FUNCTION_BLOCK ChanRcvBool (* Composite Function Block Type *)
  (* Standard: 61499-2 *)
  (* Version 0.0, 12/6/2023, vaatmar1, nxtControl GmBH, template *)
  PACKAGE Main;
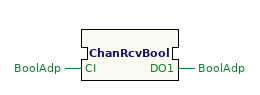
  SOCKETS
    CI : BoolAdp;
  END_SOCKETS
  PLUGS
    DO1 : BoolAdp;
  END_PLUGS
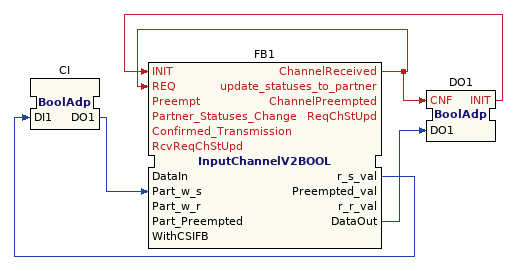
  FBS
    FB1 : InputChannelV2BOOL;
  END_FBS
  EVENT_CONNECTIONS
    DO1.INIT TO FB1.INIT;
    FB1.ChannelReceived TO DO1.CNF;
    FB1.ChannelReceived TO FB1.REQ;
  END_CONNECTIONS
  DATA_CONNECTIONS
    CI.DO1 TO FB1.Part_w_s;
    FB1.DataOut TO DO1.DO1;
    FB1.r_s_val TO CI.DI1;
  END_CONNECTIONS
END_FUNCTION_BLOCK
